// TIA Portal V16 export
// export: Created 2023-03-29T11:04:37.5273577Z, ExportSetting WithDefaults, DisplayName Totally Integrated Automation Portal, DisplayVersion V16 Update 6, DisplayName TIA Portal Version Control Interface, DisplayVersion V16 Update 2, DisplayName TIA Portal Openness, DisplayVersion V16 Update 6, DisplayName STEP 7 Professional, DisplayVersion V16 Update 6, DisplayName STEP 7 Safety, DisplayVersion V16, DisplayName WinCC Advanced, DisplayVersion V16 Update 6
DATA_BLOCK "dbHold_Sending_TCP"   // DB114
{ S7_Optimized_Access := 'FALSE' }
VERSION : 0.1
// stored: AutoNumber true, DBAccessibleFromOPCUA true, IsOnlyStoredInLoadMemory false, IsWriteProtectedInAS false
   VAR
      Sending_Hold : Struct
         set_poziom_napełniania : Real;   // wartość zadana poziomu napełniania
         set_poziom_opróżniania : Real;   // wartość zadana poziomu opróżniania
         set_bity_sterowania_napęami_1 : Word;   // bity sterowania napędami
         set_bity_sterowania_napęami_2 : Word;   // bity sterowania napędami
         set_bity_tryb_napędów_1 : Word;   // bity sterowania przełączaniem trybów pracy
         set_bity_tryb_napędów_2 : Word;   // bity sterowania przełączaniem trybów pracy
         rez_alarm_napędów : Word;   // bity kasowania alarmów napędów
         set_strategia_sterowania : Word;   // (Bit 53.0 - Wyłączony), (Bit 53.1 - Dosilanie), (Bit 53.2 - Przetłączanie), (Bit 53.3 - Automat), (Bit 53.4 - Ręczne )
         set_sterowanie_cyklem : Word;   // (Bit 55.0 - Cykl wyłączony (Bit 55.1 - Cykl dobowy), (Bit 55.2 - Cykl tygodniowy), (Bit 55.3 - Cykl ręczny)
         set_położenie_Z10 : Word;   // zadane położenie procentowe Z10
         komunikacjaPLC : Word := 1;   // kontrola komunikacji wysyłanie -> 1
         instHourStart_Filling : Int := 0;   // Godzina start napełniania
         instMinutStart_Filling : Int := 5;   // Minuta start napełniania
         instHourStop_Filling : Int := 17;   // Godzina stop napełniania
         instMinutStopt_Filling : Int := 0;   // Minuta stop napełniania
         instHourStart_City : Int := 18;   // Godzina start przetłaczanie miasto DN225
         instMinutStart_City : Int := 0;   // Minuty start przetłaczanie miasto DN225
         instHourStop_City : Int := 23;   // Godzina stop przetłaczanie miasto DN225
         instMinutStopt_City : Int := 59;   // Minuty stop przetłaczanie miasto DN225
         instHourStart_Replen : Int := 18;   // Godzina start przetłaczanie magistrala DN500
         instMinutStart_Replen : Int := 0;   // Minuty start przetłaczanie magistrala DN500
         instHourStop_Replen : Int := 23;   // Godzina stop przetłaczanie magistrala DN500
         instMinutStopt_Replen : Int := 59;   // Minuty stop przetłaczanie magistrala DN500
      END_STRUCT;
   END_VAR
BEGIN
END_DATA_BLOCK
